PROGRAM MAIN
VAR
	fbOpticalSensor : FB_OpticalSensor;
	eState : (INIT, IDLE, PUBLISH) := INIT;
	
	//BOOL Wert für Zustandsmaschine
	bEntry : BOOL := TRUE;
	bPublish : BOOL;
	
	//Instanz von Bausteine: JsonXML
	fbJsonSaxWriter : FB_JsonSaxWriter;
	
	//Instanz von selbst erstellte FB basiert auf FB von Tc3_IotBase(Publish)
	fbMqttClient : FB_MqttClient;
	
	//Instanz von selbst erstellte FB basiert auf FB von Tc3_IotBase(Subscribe)
	fbMqttSubClient : FB_MqttSubClient;
	fbMessageQueue : FB_IotMqttMessageQueue;
	fbMessage : FB_IotMqttMessage;
	
	//Struct von Verbindungsdetails, nur einmal in INIT durchgeführt
	stMqttConnect : ST_MqttConnect;
	//Payload String
	sPayload : STRING;
END_VAR

CASE eState OF
	INIT:
		//ENTRY
		bEntry := FALSE;
		
		//DO
		stMqttConnect.sClientID := 'Laptop Hazim';
		stMqttConnect.sHostName := '192.168.2.103';
		stMqttConnect.sTopicPrefix := '';
		stMqttConnect.nHostPort := 1883;
		stMqttConnect.nKeepAlive := 60;

		//EXIT
		bEntry := TRUE;
		eState := IDLE;
	
	IDLE:
		//ENTRY
		bEntry := FALSE;
		
		//DO
		fbMqttSubClient(stMqttConnect := stMqttConnect,TopicToSubscribe := 'Hazim/Mqtt Logger/Optical Sensor/Get Data',fbMqttMessage := fbMessage, fbMqttMessageQueue := fbMessageQueue); //Verbindung mit Broker Zyklisch herstellen
		//EXIT
		IF fbMqttSubClient.bGetValue THEN
			bEntry := TRUE;
			eState := PUBLISH;
		END_IF
 
	PUBLISH:
		//ENTRY
		bEntry := FALSE;
		
		//DO
		fbMqttClient(stMqttConnect := stMqttConnect); //Verbindung mit Broker Zyklisch herstellen
		//Verbindung mit Broker für Subscription auch in dieser Zustand notwendig
		fbMqttSubClient(stMqttConnect := stMqttConnect,TopicToSubscribe := 'Hazim/Mqtt Logger/Optical Sensor/Get Data',fbMqttMessage := fbMessage, fbMqttMessageQueue := fbMessageQueue); //Verbindung mit Broker Zyklisch herstellen
		
		fbOpticalSensor(); //Zyklische Aufruf der Sensor Funktonsbausteine
		
		//Json Object Erstellen und als Json String übergeben
		fbJsonSaxWriter.ResetDocument();
		fbJsonSaxWriter.StartObject();
		fbJsonSaxWriter.AddKeyDateTime('Timestamp',F_GetTime());
		fbJsonSaxWriter.AddKeyNumber('Distance',fbOpticalSensor.nDistance);
		fbJsonSaxWriter.AddKeyBool('Distance Range Check',fbOpticalSensor.bValueRangeCheck);
		fbJsonSaxWriter.EndObject();
		sPayload := fbJsonSaxWriter.GetDocument();
		
		//Zu MQTT Broker Publish
		fbMqttClient.Publish(sPublishTopic := 'Hazim/Mqtt Logger/Optical Sensor',sPayload := sPayload);
		
		//EXIT
		IF NOT fbMqttSubClient.bGetValue THEN
			bEntry := TRUE;
			eState := IDLE;
		END_IF
		
END_CASE

END_PROGRAM

(* stored: Version 1.1.0.1, ProductVersion 3.1.4024.15
   POU MAIN: Id {7453db33-6c9d-480b-b7d3-811b216897b1}, SpecialFunc None *)
